FUNCTION proj1_TupleStruct_2: DINT
{ S7_Optimized_Access := 'true' }
    VAR_INPUT
        tuple: TupleStruct_2;
    END_VAR

BEGIN
    proj1_TupleStruct_2 := tuple.field1;
END_FUNCTION
